Staubli VAL3: Form_MainS.pgx

public program Form_MainS(string x_sBottomList)
  local num l_nIndex
  local bool l_bRes
  local string l_sBuff[20]
begin
  //把字符串给分开，使用,作为分隔符
  //主界面
  call Str_SplitComma(l_bRes,x_sBottomList,l_sBuff)
  if !l_bRes
    return
  endIf
   call Form_Main(l_sBuff)
end
